// TIA Portal V20 export
DATA_BLOCK "Process_Control_DB"   // DB98
// stored: InstanceOfName Process_Control, InstanceOfType FB
"Process_Control"
   // VAR_INPUT
   //    Level : Real;
   // END_VAR
BEGIN
END_DATA_BLOCK
